FUNCTION_BLOCK POU
VAR_INPUT
END_VAR
VAR_OUTPUT
END_VAR
VAR
END_VAR

// NETWORK 1

END_FUNCTION_BLOCK

(* stored: Version 1.1.0.1, ProductVersion 3.1.4024.2
   POU POU: Id {9e510904-31e3-464e-9503-0b4c4916ac8c}, SpecialFunc None *)
